PROGRAM Stn053_10_EvalLnSwPrestopGrn
VAR
	{attribute 'TcLinkToOSO' := '.iPuckPresent := <0,1,1>TIIB[N32S00 (AL1332)]^N32S01 (AL2341)^TxPDO^input byte 0;
		.oStopLower :=  <0,1,3>TIIB[N32S00 (AL1332)]^N32S02 (EX260)^RxPDO^output byte 0'}
	fbConvStop: FB_ConvStop;
END_VAR

//  This code instantiates a component that is implimented as a common function block
//    Note that I/O is linked directly to I/O variables inside the named instance

gStn053_10_EvalLnSwPrestopGrn.ConvRunning := gStn053_16_EvalLnSw.BoschInfeedConvRunning;

fbConvStop(
	pStn := ADR(gStn053),
	pCmp := ADR(gStn053_10_EvalLnSwPrestopGrn),
	pUpstreamStop := 0,
	pStateTraceBuffer := ADR(gStn053_StateTraceBuffer),
	pStateTraceFifo := ADR(gStn053_StateTraceFifo),
	pStats := ADR(gStn053_02_Stats));

END_PROGRAM

(* stored: Version 1.1.0.1, ProductVersion 3.1.4024.6
   POU Stn053_10_EvalLnSwPrestopGrn: Id {0439e43a-aff8-4bbe-8ca0-2c83b4bcd036}, SpecialFunc None *)
